PROGRAM READ_POS
VAR
	MC_ReadActualPosition1 : MC_ReadActualPosition;
	MC_ReadActualPosition2 : MC_ReadActualPosition;
	MC_ReadActualPosition3 : MC_ReadActualPosition;
	MC_ReadActualPosition4 : MC_ReadActualPosition;
END_VAR

MC_ReadActualPosition1(
	Axis:= AXIS.Axis1, 
	Enable:= , 
	Valid=> , 
	Busy=> , 
	Error=> , 
	ErrorID=> , 
	Position=> );
	
MC_ReadActualPosition2(
	Axis:= AXIS.Axis2, 
	Enable:= , 
	Valid=> , 
	Busy=> , 
	Error=> , 
	ErrorID=> , 
	Position=> );
	
MC_ReadActualPosition3(
	Axis:= AXIS.Axis3, 
	Enable:= , 
	Valid=> , 
	Busy=> , 
	Error=> , 
	ErrorID=> , 
	Position=> );
	
MC_ReadActualPosition4(
	Axis:= AXIS.Axis4, 
	Enable:= , 
	Valid=> , 
	Busy=> , 
	Error=> , 
	ErrorID=> , 
	Position=> );

END_PROGRAM

(* stored: Version 1.1.0.1, ProductVersion 3.1.4024.0
   POU READ_POS: Id {ead86361-caf5-43c4-a7c8-e87af4056d28}, SpecialFunc None *)
